{attribute addProperty BoxType "KL9191"}
{attribute addProperty Id "Channel_1Channel_89E8594300"}
{attribute addProperty CRC "895822927"}
{attribute addProperty SizeInBites "0"}
{attribute addProperty SizeInBytes "0"}
TYPE KL9191_35652C4F :
STRUCT
	{attribute addProperty Name "Channel_1"}
	Channel_1 : Channel_89E85943;
END_STRUCT
END_TYPE

(* stored: Version 1.2.0.0, ProductVersion 3.1.4024.9
   DUT KL9191_35652C4F: Id {33efa9e0-ba1e-4a33-931a-69179623288a} *)
